PROGRAM PRG_OPT
VAR
    bInit: BOOL := TRUE;
    fbMotionRxG: FB_MotionStage;
    fbMotionXG: FB_MotionStage;
    fbMotionRzPM: FB_MotionStage;
END_VAR


//Lock stages until they are tested
Main.M10.nEnableMode := ENUM_StageEnableMode.NEVER ;
Main.M11.nEnableMode := ENUM_StageEnableMode.NEVER ;
Main.M14.nEnableMode := ENUM_StageEnableMode.NEVER ;

IF bINIT THEN

    Main.M10.nBrakeMode := ENUM_StageBrakeMode.NO_BRAKE;
    Main.M10.bHardwareEnable := TRUE;
    Main.M10.bPowerSelf := TRUE;
    Main.M11.nBrakeMode := ENUM_StageBrakeMode.NO_BRAKE;
    Main.M11.bHardwareEnable := TRUE;
    Main.M11.bPowerSelf := TRUE;
    Main.M14.nBrakeMode := ENUM_StageBrakeMode.NO_BRAKE;
    Main.M14.bHardwareEnable := TRUE;
    Main.M14.bPowerSelf := TRUE;

    Main.M10.nEnableMode := ENUM_StageEnableMode.DURING_MOTION ;
    Main.M11.nEnableMode := ENUM_StageEnableMode.DURING_MOTION ;
    Main.M14.nEnableMode := ENUM_StageEnableMode.DURING_MOTION ;

    bINIT := FALSE;
END_IF;


fbMotionRxG(stMotionStage:= Main.M10);
fbMotionXG(stMotionStage:= Main.M11);
fbMotionRzPM(stMotionStage:= Main.M14);

END_PROGRAM

(* stored: Version 1.1.0.1, ProductVersion 3.1.4022.18
   POU PRG_OPT: Id {9fd4ef96-d0b3-4d92-a155-89dc0eb4c6d2}, SpecialFunc None *)
